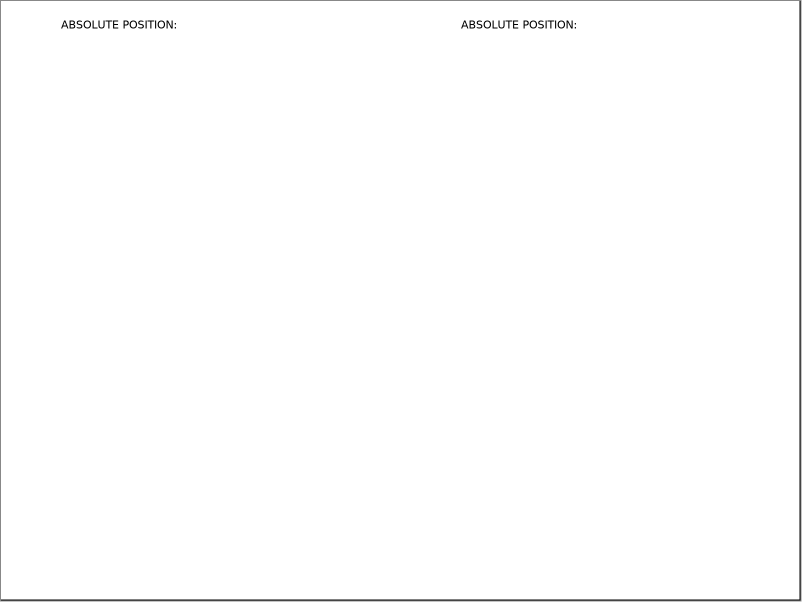
VISUALIZATION F46_Phasing_Relative  // 802x602
    Rectangle (0,0 800x600)
    Label (10,10 170x30), "ABSOLUTE POSITION:"
    Label (410,10 170x30), "ABSOLUTE POSITION:"
END_VISUALIZATION

(* stored: Version 1.1.0.1, ProductVersion 3.1.4022.7
   Visu F46_Phasing_Relative: Id {98c54993-9514-4e4f-a76c-884bca84d879} *)
